TYPE DANCERCONTROL_ERRORS :
(
	DANCERCONTROL_ERROR_INVALID_POINTER := 16#4B50,
	DANCERCONTROL_ERROR_INVALID_PID_PARAMETER := 16#4B51,
	DANCERCONTROL_ERROR_INVALID_CYCLETIME := 16#4B52
) UDINT;
END_TYPE

(* stored: Version 1.1.0.1, ProductVersion 3.1.4024.11
   DUT DANCERCONTROL_ERRORS: Id {a1e06fde-61cc-4dd2-9464-c6146f8f824d} *)
